// Mitsubishi GX Works2 project: 13   PLC: FX2N/FX2NC

PROGRAM MAIN
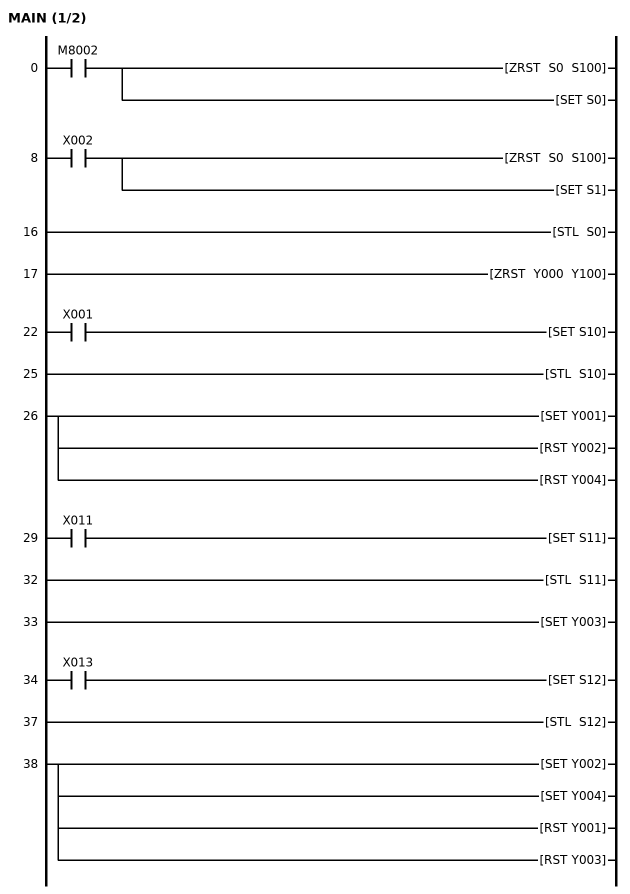
0     LD      M8002
      ZRST    S0 S100
      SET     S0
8     LD      X002
      ZRST    S0 S100
      SET     S1
16    STL     S0
17    ZRST    Y000 Y100
22    LD      X001
      SET     S10
25    STL     S10
26    SET     Y001
      RST     Y002
      RST     Y004
29    LD      X011
      SET     S11
32    STL     S11
33    SET     Y003
34    LD      X013
      SET     S12
37    STL     S12
38    SET     Y002
      SET     Y004
      RST     Y001
      RST     Y003
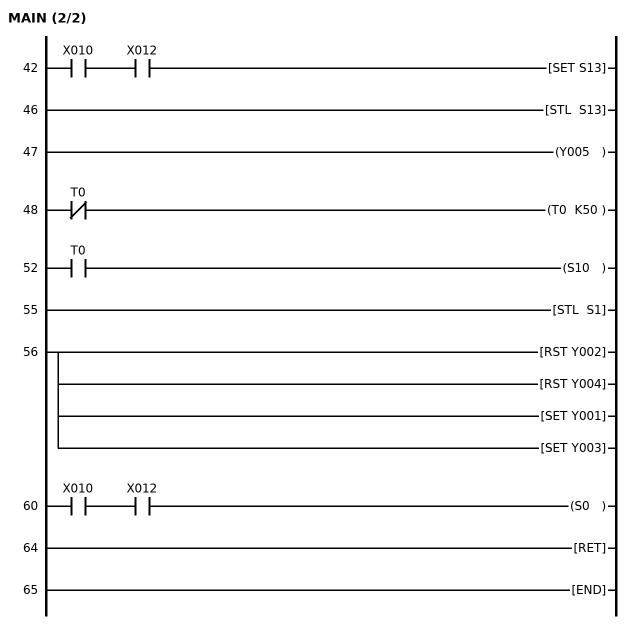
42    LD      X010
      AND     X012
      SET     S13
46    STL     S13
47    OUT     Y005
48    LDI     T0
      OUT     T0 K50
52    LD      T0
      OUT     S10
55    STL     S1
56    RST     Y002
      RST     Y004
      SET     Y001
      SET     Y003
60    LD      X010
      AND     X012
      OUT     S0
64    RET
65    END
END_PROGRAM

// device comments not shown above
BL0  ; main
BL1  ; a
BL2  ; b
